% RSLogix 500 project test 22222.RSS, saved by version 8.30.00.15 %
PROJECT "UNTITLED"    % processor: MicroLogix 1000 %

PROGRAM FILES
  LAD 2 "MAIN_PROG"  6 rungs
  LAD 3 "USER_FAULT"  1 rungs
  LAD 4 "HSC_INT"  1 rungs
  LAD 5 "STI_INT"  1 rungs
  LAD 6, 7, 8, 9, 10, 11, 12, 13, 14, 15, 16: only END

DATA FILES
  O0 OUTPUT  1 elements
  I1 INPUT  2 elements
  S2 STATUS  33 elements
  B3 BINARY  32 elements
  T4 TIMER  40 elements
  C5 COUNTER  32 elements
  R6 CONTROL  16 elements
  N7 INTEGER  105 elements

LADDER 2 "MAIN_PROG"
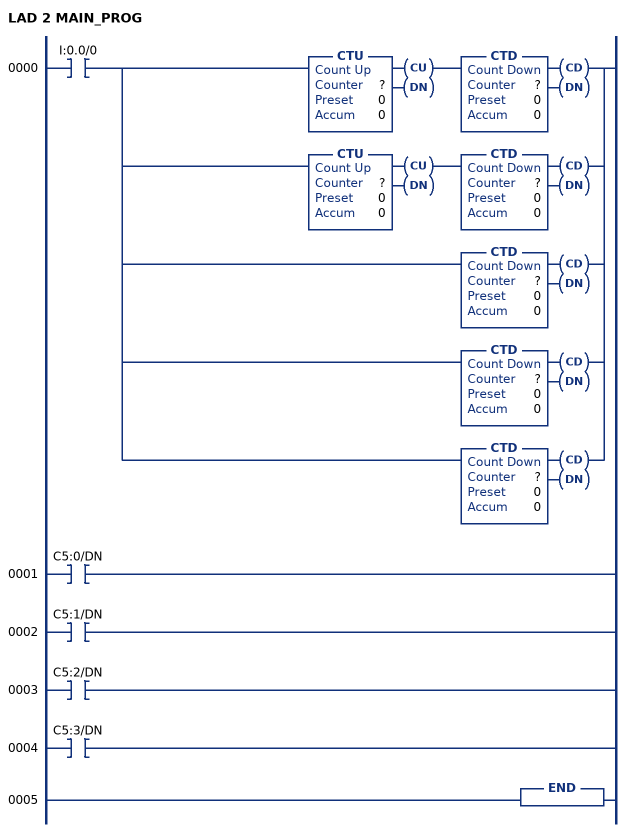
% Rung: 0 %  % edit flag set %
SOR XIC I:0.0/0 BST BST BST BST CTU ? 0 0 CTD ? 0 0 NXB CTU ? 0 0 CTD ? 0 0 BND NXB CTD ? 0 0 BND NXB CTD ? 0 0 BND NXB CTD ? 0 0 BND EOR
% Rung: 1 %  % edit flag set %
SOR XIC C5:0/DN EOR
% Rung: 2 %  % edit flag set %
SOR XIC C5:1/DN EOR
% Rung: 3 %  % edit flag set %
SOR XIC C5:2/DN EOR
% Rung: 4 %  % edit flag set %
SOR XIC C5:3/DN EOR
% Rung: 5 %
SOR END EOR

DATA TABLE (non-zero values as saved)
DATA C5
% .PRE .ACC %
% C5:0 % 1 0
% C5:1 % 2 0
% C5:2 % 3 0
% C5:3 % 4 0
% C5:4 % 5 0
% C5:5 % 0 1
% C5:6 % 0 1
% C5:7 % 0 1
% C5:8 % 0 1
